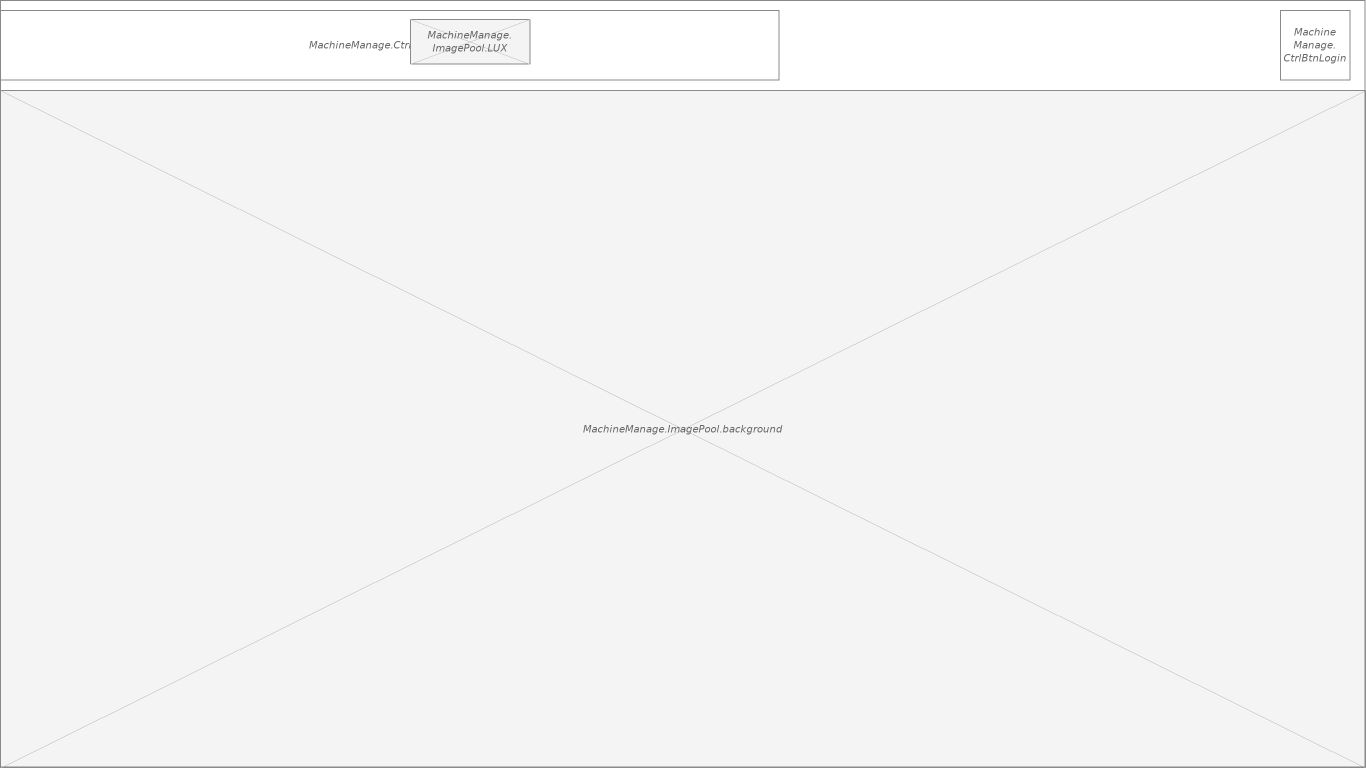
VISUALIZATION FrameMain  // 1366x768
    Frame (0,10 779x70)
        shows MachineManage.CtrlPageSwitch(System := G_stSystem)
    Image (0,90 1366x678), image: MachineManage.ImagePool.background
    Frame (1280,10 70x70)
        shows MachineManage.CtrlBtnLogin()
    Rectangle (422,27 100x30)
    Image (410,19 120x45), image: MachineManage.ImagePool.LUX
END_VISUALIZATION

(* stored: Version 1.1.0.1, ProductVersion 3.1.4024.3
   Visu FrameMain: Id {4725c32d-0c37-422a-9c45-1d9e29bdb5bc} *)
